// TIA Portal V16 export
// export: Created 2021-09-20T14:24:38.1290246Z, ExportSetting WithDefaults, DisplayName Totally Integrated Automation Portal, DisplayVersion V16 Update 1, DisplayName TIA Portal Version Control Interface, DisplayVersion V16, DisplayName TIA Portal Openness, DisplayVersion V16, DisplayName SINAMICS Startdrive Advanced, DisplayVersion V16 Update 5, DisplayName SINAMICS Startdrive G130, G150, S120, S150, SINAMICS MV, S210, DisplayVersion V16 Update 5, DisplayName SINAMICS Startdrive G110M, G120, G120C, G120D, G120P, G115D, DisplayVersion V16 Update 5, DisplayName STEP 7 Professional, DisplayVersion V16, DisplayName STEP 7 Safety, DisplayVersion V16, DisplayName WinCC Professional, DisplayVersion V16
DATA_BLOCK "Data_block_1"   // DB1
{ S7_Optimized_Access := 'TRUE' }
VERSION : 0.1
// stored: AutoNumber true, DBAccessibleFromOPCUA true, IsOnlyStoredInLoadMemory false, IsRetainMemResEnabled false, IsWriteProtectedInAS false, MemoryReserve 100
   VAR
      ex : Bool;
      ex_1 : Bool;
      ex_2 : Bool;
      ex_3 : Bool;
      ex_4 : Bool;
      ex_5 : Bool;
      ex_6 : Bool;
      ex_7 : Bool;
      ex_8 : Bool;
      ex_9 : Bool;
      new : Bool;
      new_1 : Bool;
      new_2 : Bool;
   END_VAR
BEGIN
END_DATA_BLOCK
